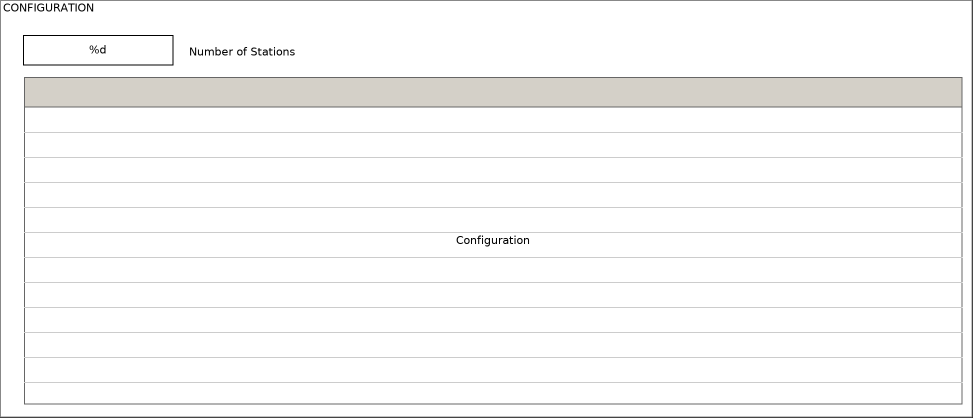
VISUALIZATION VI_XTSStationsConfigurationVisu  // 973x418
VAR_IN_OUT
	xts : XTS_System;
END_VAR
VAR
	stTableStruct : ARRAY [1..25] OF stTableStructx10;
END_VAR
    Rectangle (0,0 973x418), "CONFIGURATION"
    Table (24,77 938x327), "Configuration", data array: stTableStruct
        p3854506369: xts.stCfg.stStationsCfg[INDEX].sName
        p1892666644: xts.stCfg.stStationsCfg[INDEX].lrStartPosition
        p338671338: xts.stCfg.stStationsCfg[INDEX].lrStopPosition[1]
        p2170511999: xts.stCfg.stStationsCfg[INDEX].lrStopPosition[2]
        p3723444502: xts.stCfg.stStationsCfg[INDEX].lrStopPosition[3]
        p1218418051: xts.stCfg.stStationsCfg[INDEX].lrProcessingTime
        p746581629: xts.stCfg.stStationsCfg[INDEX].uiNumStopPositions
        p3104783080: xts.stCfg.stStationsCfg[INDEX].lrTravelTime
        p7306298: xts.stCfg.stStationsCfg[INDEX].lrEndPosition
        p511219082: Start Position
        p1755163831: Stop Position 1
        p4092479075: Stop Position 2
        p2237128397: Stop Position 3
        p505689113: Process Time
        p1757482276: Stop Positions
        p4088588272: Travel Time
        p2243050616: Extra Cfg.
        p516019884: End Position
        p2685023577: stTableStruct.b1
        p3312258591: stTableStruct.b2
        p1791247317: stTableStruct.b3
        p262371475: stTableStruct.b4
        p4008173056: stTableStruct.b5
        p2340480326: stTableStruct.b6
        p606709900: stTableStruct.b7
        p1095668682: stTableStruct.b8
        p1037165547: stTableStruct.b9
        p1488378029: stTableStruct.b10
        Columns.Column.[3].Template: OnMouseClick: write the text variable via Default
        Columns.Column.[6].Template: OnMouseClick: write the text variable via Default, min 1, max 3
        Columns.Column.[4].Template: OnMouseClick: write the text variable via Default
        Columns.Column.[5].Template: OnMouseClick: write the text variable via Default
        Columns.Column.[2].Template: OnMouseClick: write the text variable via Default
        Columns.Column.[0].Template: OnMouseClick: write the text variable via Default
        Columns.Column.[1].Template: OnMouseClick: write the text variable via Default
        Columns.Column.[7].Template: OnMouseClick: write the text variable via Default
        Columns.Column.[9].Template: OnMouseClick: write the text variable via Default
    Label (186,37 150x30), "Number of Stations"
    Rectangle (23,35 150x30), "%d", text variable: xts.stCfg.udiNumStations
        OnMouseClick: write the text variable via Default
END_VISUALIZATION

(* stored: Version 1.1.0.1, ProductVersion 3.1.4024.11
   Visu VI_XTSStationsConfigurationVisu: Id {8c33ed62-29e5-4c4a-8bc8-2674a2df4738} *)
